(* CoDeSys 2.3.9.35 project: Q4_SISTEMA_DE_ESTEIRA_(COM MODELO).pro *)
(* Author: Altus *)
(* Libraries: DU35x.lib 7.7.11 15:59:13, Navigation.lib 15.7.11 10:06:00, SysLibTargetVisu.lib 26.11.08 09:53:28, Standard.lib 26.11.08 09:46:20, Iecsfc.lib 26.11.08 09:46:14, SYSLIBCALLBACK.LIB 26.11.08 09:53:30 *)

(* PLC configuration (modules and I/O channels)
Configuração do CP [Root] node -1, in %IB0 out %QB0
  Comunicação [Comunica] node 0, in %IB0 out %QB0
    COM1 [COM1] node 0, in %IB0 out %QB0 {BaudRate = 115200; Paridade = Sem Paridade; StopBits = 1 Stop Bit; Modem = Sem RTS/CTS; Delay = 5}
      MToolIEC [Codesys] node 0, in %IB0 out %QB0
    COM2 [COM2] node 1, in %IB0 out %QB0 {BaudRate = 115200; Paridade = Sem Paridade; StopBits = 1 Stop Bit; Modem = Sem RTS/CTS; Delay = 5}
      Desabilitada [Desabilitado485] node 0, in %IB0 out %QB0
  Barramento [Barramento] node 1, in %IB0 out %QB0
    Entradas [Entradas] node 0, in %IB0 out %QB0
      Entradas Digitais 0 [Entradas0] node 0, in %IW0 out %QB0
        I00 AT %IX0.0 [BitInput] I0.0
        I01 AT %IX0.1 [BitInput] I0.1
        I02 AT %IX0.2 [BitInput] I0.2
        I03 AT %IX0.3 [BitInput] I0.3
        I04 AT %IX0.4 [BitInput] I0.4
        I05 AT %IX0.5 [BitInput] I0.5
        I06 AT %IX0.6 [BitInput] I0.6
        I07 AT %IX0.7 [BitInput] I0.7
        I08 AT %IX0.8 [BitInput] I0.8
      Entradas Digitais 1 [Entradas1] node 0, in %IW1 out %QB0
        I10 AT %IX1.0 [BitInput] I1.0
        I11 AT %IX1.1 [BitInput] I1.1
        I12 AT %IX1.2 [BitInput] I1.2
        I13 AT %IX1.3 [BitInput] I1.3
        I14 AT %IX1.4 [BitInput] I1.4
        I15 AT %IX1.5 [BitInput] I1.5
        I16 AT %IX1.6 [BitInput] I1.6
        I17 AT %IX1.7 [BitInput] I1.7
        I18 AT %IX1.8 [BitInput] I1.8
      Entradas Digitais 2 [Entradas2] node 0, in %IW2 out %QB0
        I20 AT %IX2.0 [BitInput] I2.0
        I21 AT %IX2.1 [BitInput] I2.1
      Entradas Analógicas [EntradaAnalogica] node 0, in %IW4 out %QB0
        AI0 AT %IW4 [WordInput] AI0 {TipoAnalogica = Channel Disable; FiltroAnalogica = Filter 0 - AI=2ms  / AV=90ms; FundoEscala = 0}
        AI1 AT %IW5 [WordInput] AI1 {TipoAnalogica = Channel Disable; FiltroAnalogica = Filter 0 - AI=2ms  / AV=90ms; FundoEscala = 0}
        AI2 AT %IW6 [WordInput] AI2 {TipoAnalogica = Channel Disable; FiltroAnalogica = Filter 0 - AI=2ms  / AV=90ms; FundoEscala = 0}
        AI3 AT %IW7 [WordInput] AI3 {TipoAnalogica = Channel Disable; FiltroAnalogica = Filter 0 - AI=2ms  / AV=90ms; FundoEscala = 0}
      Entradas Rápidas [EntradasRapidas] node 1, in %IB16 out %QB0
        Bloco 0 [Bloco0] node 0, in %IB16 out %QB0
          Desabilitado [DesabilitadoBloco0] node 0, in %IB16 out %QB0
        Bloco 1 [Bloco1] node 1, in %IB16 out %QB0
          Desabilitado [DesabilitadoBloco1] node 0, in %IB16 out %QB0
        Entrada Configuravél Bloco 0 [EntradaConfiBloco0] node 2, in %IB16 out %QB0
          Contador 0 [EntradaConfContador0] node 0, in %IB16 out %QB0 {EntradaConfiguravelContador = Disable}
        Entrada Configuravél Bloco 1 [EntradaConfiBloco1] node 3, in %IB16 out %QB0
          Contador 2 [EntradaConfContador2] node 0, in %IB16 out %QB0 {EntradaConfiguravelContador = Disable}
    Saídas [Saidas] node 1, in %IB13 out %QB0
      Saídas Digitais 0 [Saidas0] node 0, in %IW0 out %QW0
        Q00 AT %QX0.0 [BitOutput] Q0.0
        Q01 AT %QX0.1 [BitOutput] Q0.1
        Q02 AT %QX0.2 [BitOutput] Q0.2
        Q03 AT %QX0.3 [BitOutput] Q0.3
        Q04 AT %QX0.4 [BitOutput] Q0.4
        Q05 AT %QX0.5 [BitOutput] Q0.5
        Q06 AT %QX0.6 [BitOutput] Q0.6
        Q07 AT %QX0.7 [BitOutput] Q0.7
      Saídas Digitais 1 [Saidas1] node 0, in %IW0 out %QW1
        Q10 AT %QX1.0 [BitOutput] Q1.0
        Q11 AT %QX1.1 [BitOutput] Q1.1
        Q12 AT %QX1.2 [BitOutput] Q1.2
        Q13 AT %QX1.3 [BitOutput] Q1.3
        Q14 AT %QX1.4 [BitOutput] Q1.4
        Q15 AT %QX1.5 [BitOutput] Q1.5
        Q16 AT %QX1.6 [BitOutput] Q1.6
        Q17 AT %QX1.7 [BitOutput] Q1.7
      Saídas Analógicas [SaidaAnalogica] node 0, in %IW0 out %QW3
        AO0 AT %QW3 [WordOutput] AO0 {TipoAnalogica = Channel Disable; FundoEscala = 0}
        AO1 AT %QW4 [WordOutput] AO1 {TipoAnalogica = Channel Disable; FundoEscala = 0}
      Saídas Rápidas [SaidasRapidas] node 1, in %IB0 out %QB10
        Saída Rápida 0 Desabilitada [DesabilitadoF0] node 0, in %IB0 out %QB10
        Saída Rápida 1 Desabilitada [DesabilitadoF1] node 1, in %IB0 out %QB10
      Saídas Comum de Contador [SaidasContador] node 2, in %IB0 out %QB10
        Saída do Bloco 0 Desabilitada [DesabilitadoSaidaBloco0] node 0, in %IB0 out %QB10
        Saída do Bloco 1 Desabilitada [DesabilitadoSaidaBloco1] node 1, in %IB0 out %QB10
  Eventos Externos [Eventos] node 2, in %IB13 out %QB6
    Evento Temporizado [TimerEvent] node 0, in %IB13 out %QB6 {Intervalo = 10}
*)

(* Task configuration *)
TASK PRINCIPAL (PRIORITY := 1, INTERVAL := T#1ms);
	PLC_PRG();
END_TASK
TASK NAVIGATION (PRIORITY := 1, INTERVAL := T#20ms);
	NAVEGA();
END_TASK
TASK VISUALIZATION (PRIORITY := 1, INTERVAL := T#500ms);
	MAINTARGETVISU_PAINT_CODE
END_TASK
TASK KEYBOARD_USAGE (PRIORITY := 1, INTERVAL := T#20ms);
	MAINTARGETVISU_INPUT_CODE
END_TASK

(* POU PLC_PRG, LD *)
PROGRAM PLC_PRG
VAR
    (* ========================================================= *)
    (* ENTRADAS FISICAS (Chaves e Sensores - %IX)             *)
    (* ========================================================= *)
    a0 AT %IX0.0: BOOL; (* Sensor de Fim de Curso: Cilindro A Recuado *)
    a1 AT %IX0.1: BOOL; (* Sensor de Fim de Curso: Cilindro A Avancado *)
    b0 AT %IX0.2: BOOL; (* Sensor de Fim de Curso: Cilindro B Recuado *)
    b1 AT %IX0.3: BOOL; (* Sensor de Fim de Curso: Cilindro B Avancado *)
    c0 AT %IX0.4: BOOL; (* Sensor de Fim de Curso: Cilindro C Recuado *)
    c1 AT %IX0.5: BOOL; (* Sensor de Fim de Curso: Cilindro C Avancado *)
    CH AT %IX0.6: BOOL; (* Chave de Controle de Ciclo S *)
    SP AT %IX0.7: BOOL; (* Sensor de Presenca de Embalagem Sp - NF *)

    (* ========================================================= *)
    (* SAIDAS FISICAS (Atuadores - %QX)                       *)
    (* ========================================================= *)
    CA AT %QX1.0: BOOL; (* Comando: Valvula do Cilindro A *)
    CB AT %QX1.1: BOOL; (* Comando: Valvula do Cilindro B *)
    CC AT %QX1.2: BOOL; (* Comando: Valvula do Cilindro C *)
    M  AT %QX1.3: BOOL; (* Comando: Motor de acionamento da esteira *)

    (* ========================================================= *)
    (* ESTADOS DO AFD (Memorias de Etapa - %MX1.x)            *)
    (* ========================================================= *)
    S0 AT %MX1.0: BOOL; (* Estado 0: Repouso / Espera de embalagem *)
    S1 AT %MX1.1: BOOL; (* Estado 1: Avancar Cilindro A *)
    S2 AT %MX1.2: BOOL; (* Estado 2: Avancar Cilindro B *)
    S3 AT %MX1.3: BOOL; (* Estado 3: Recuar Cilindro C e Dosagem *)
    S4 AT %MX1.4: BOOL; (* Estado 4: Avancar Cilindro C *)
    S5 AT %MX1.5: BOOL; (* Estado 5: Recuar A e B simultaneamente *)
    S6 AT %MX1.6: BOOL; (* Estado 6: Esperar saida da embalagem cheia *)
    S_erro AT %MX1.7: BOOL; (* Estado Erro: Seguranca e Intertravamento *)

    (* ========================================================= *)
    (* TRANSICOES DO AFD (Condicoes de Disparo - %MX2.x e %MX3.x)*)
    (* ========================================================= *)
    T0 AT %MX2.0: BOOL; (* Disparo da transicao de S0 para S1 *)
    T1 AT %MX2.1: BOOL; (* Disparo da transicao de S1 para S2 *)
    T2 AT %MX2.2: BOOL; (* Disparo da transicao de S2 para S3 *)
    T3 AT %MX2.3: BOOL; (* Disparo da transicao de S3 para S4 *)
    T4 AT %MX2.4: BOOL; (* Disparo da transicao de S4 para S5 *)
    T5 AT %MX2.5: BOOL; (* Disparo da transicao de S5 para S6 *)
    T6 AT %MX2.6: BOOL; (* Disparo da transicao de S6 para S0 *)
    TE AT %MX3.2: BOOL; (* Disparo da transicao Global de Falha para S_erro *)
    TR AT %MX3.1: BOOL; (* Disparo da transicao de Retorno para S0 *)

    (* ========================================================= *)
    (* VARIAVEIS INTERNAS DE CONTROLO E SINALIZACAO           *)
    (* ========================================================= *)
    F      AT %MX0.6: BOOL; (* Flag: Condicao Global de Falha Ativa *)
    RESET  AT %MX3.0: BOOL; (* Comando/Flag de Reset de Erro *)
    ALARME AT %MX3.4: BOOL; (* Sinalizacao de Alarme / Intertravamento *)

    (* ========================================================= *)
    (* BLOCO FUNCIONAL: TEMPORIZADOR (Dosagem)                *)
    (* ========================================================= *)
    TEMPORIZADOR1: TON;     (* Instancia do Bloco Timer On-Delay *)
    T1_EN AT %MX0.2: BOOL;  (* Sinal para habilitar/iniciar a contagem do tempo *)
    QT1   AT %MX0.3: BOOL;  (* Saida de tempo esgotado 5 segundos *)

    (* ========================================================= *)
    (* BLOCO FUNCIONAL: CONTADOR (Lote de 10 Ciclos)          *)
    (* ========================================================= *)
    CTU: CTU;         (* CORRIGIDO: Nao usar CTU: CTU para evitar erro *)
    CU    AT %MX0.0: BOOL;  (* Pulso de entrada para incremento do contador *)
    QCU   AT %MX0.1: BOOL;  (* Saida indicando que o limite do lote foi atingido *)
    COUNT AT %MW10: INT;    (* Registo de memoria Word com o valor atual *)
    P: R_TRIG;              (* Bloco detetor de borda de subida Trigger *)
END_VAR
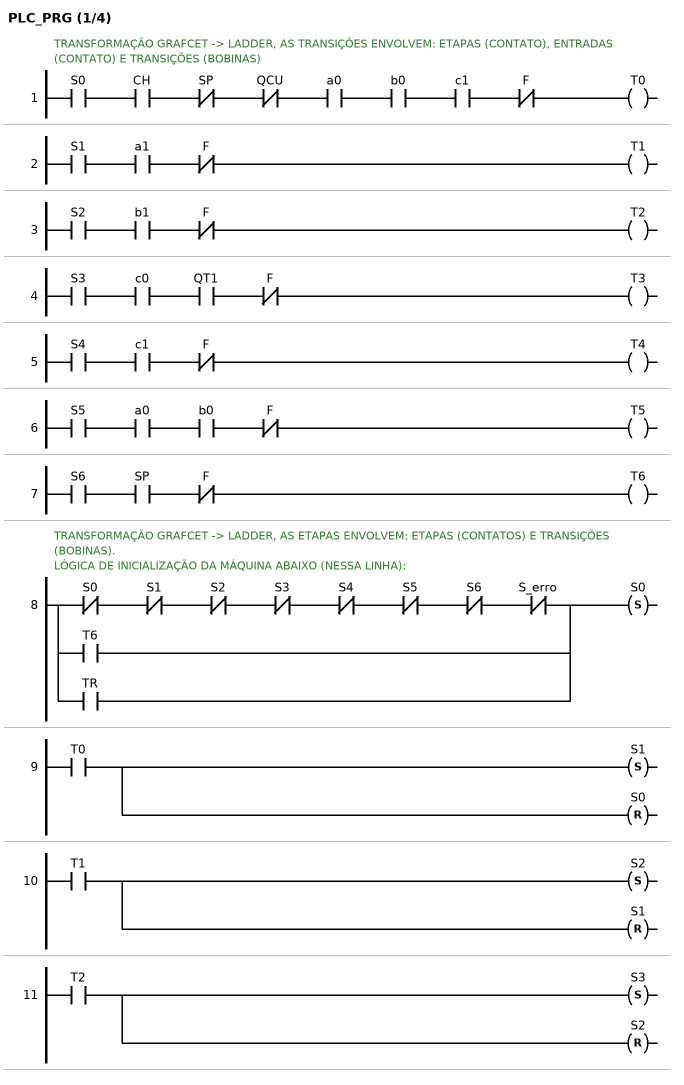
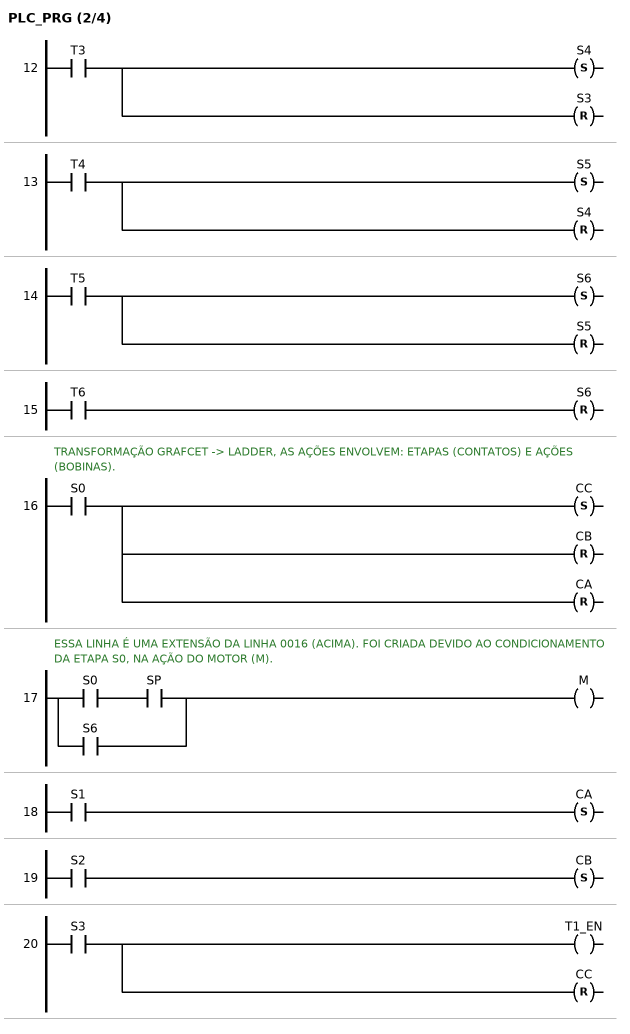
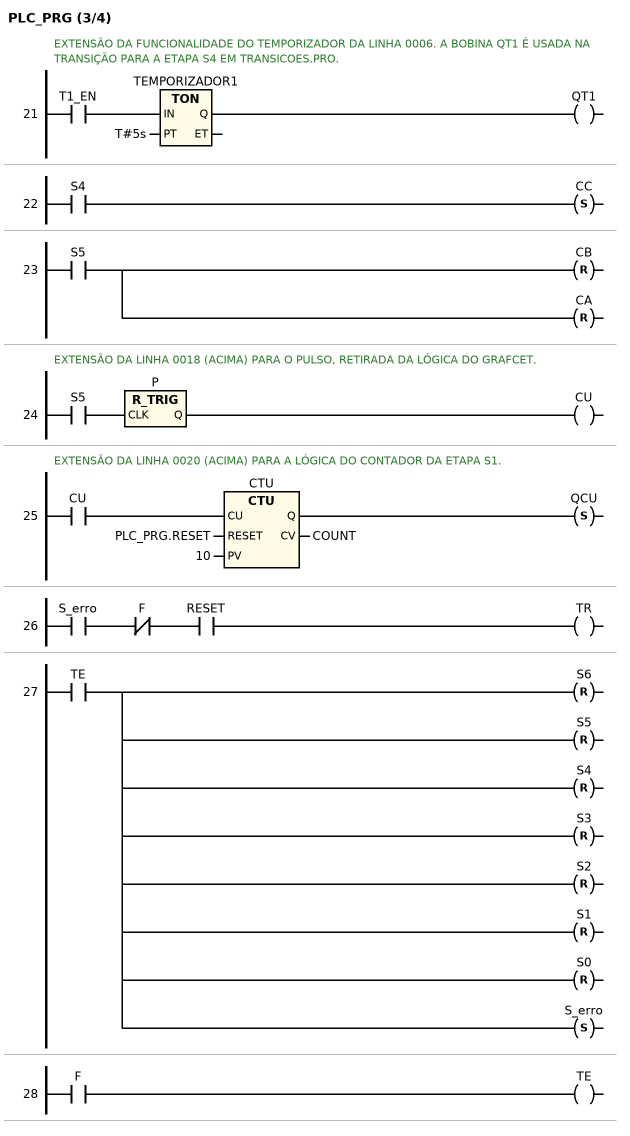
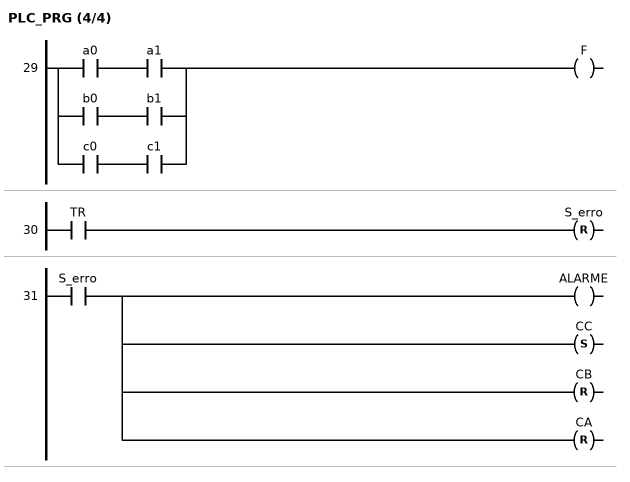
_LD_ (* Ladder Diagram *)
NETWORK 1 (* TRANSFORMAÇÃO GRAFCET -> LADDER, AS TRANSIÇÕES ENVOLVEM: ETAPAS (CONTATO), ENTRADAS (CONTATO) E TRANSIÇÕES (BOBINAS) *)
	[S0] - [CH] - [/SP] - [/QCU] - [a0] - [b0] - [c1] - [/F] --- (T0)
NETWORK 2
	[S1] - [a1] - [/F] --- (T1)
NETWORK 3
	[S2] - [b1] - [/F] --- (T2)
NETWORK 4
	[S3] - [c0] - [QT1] - [/F] --- (T3)
NETWORK 5
	[S4] - [c1] - [/F] --- (T4)
NETWORK 6
	[S5] - [a0] - [b0] - [/F] --- (T5)
NETWORK 7
	[S6] - [SP] - [/F] --- (T6)
NETWORK 8 (* TRANSFORMAÇÃO GRAFCET -> LADDER, AS ETAPAS ENVOLVEM: ETAPAS (CONTATOS) E TRANSIÇÕES (BOBINAS). / LÓGICA DE INICIALIZAÇÃO DA MÁQUINA ABAIXO (NESSA LINHA): *)
	{ [/S0] - [/S1] - [/S2] - [/S3] - [/S4] - [/S5] - [/S6] - [/S_erro] | [T6] | [TR] } --- (S S0)
NETWORK 9
	[T0] --- (S S1) (R S0)
NETWORK 10
	[T1] --- (S S2) (R S1)
NETWORK 11
	[T2] --- (S S3) (R S2)
NETWORK 12
	[T3] --- (S S4) (R S3)
NETWORK 13
	[T4] --- (S S5) (R S4)
NETWORK 14
	[T5] --- (S S6) (R S5)
NETWORK 15
	[T6] --- (R S6)
NETWORK 16 (* TRANSFORMAÇÃO GRAFCET -> LADDER, AS AÇÕES ENVOLVEM: ETAPAS (CONTATOS) E AÇÕES (BOBINAS). *)
	[S0] --- (S CC) (R CB) (R CA)
NETWORK 17 (* ESSA LINHA É UMA EXTENSÃO DA LINHA 0016 (ACIMA). FOI CRIADA DEVIDO AO CONDICIONAMENTO DA ETAPA S0, NA AÇÃO DO MOTOR (M). *)
	{ [S0] - [SP] | [S6] } --- (M)
NETWORK 18
	[S1] --- (S CA)
NETWORK 19
	[S2] --- (S CB)
NETWORK 20
	[S3] --- (T1_EN) (R CC)
NETWORK 21 (* EXTENSÃO DA FUNCIONALIDADE DO TEMPORIZADOR DA LINHA 0006. A BOBINA QT1 É USADA NA TRANSIÇÃO PARA A ETAPA S4 EM TRANSICOES.PRO. *)
	[T1_EN] - TEMPORIZADOR1:TON(IN: *, PT: T#5s) --- (QT1)
NETWORK 22
	[S4] --- (S CC)
NETWORK 23
	[S5] --- (R CB) (R CA)
NETWORK 24 (* EXTENSÃO DA LINHA 0018 (ACIMA) PARA O PULSO, RETIRADA DA LÓGICA DO GRAFCET. *)
	[S5] - P:R_TRIG(CLK: *) --- (CU)
NETWORK 25 (* EXTENSÃO DA LINHA 0020 (ACIMA) PARA A LÓGICA DO CONTADOR DA ETAPA S1. *)
	[CU] - CTU:CTU(CU: *, RESET: PLC_PRG.RESET, PV: 10, CV => COUNT) --- (S QCU)
NETWORK 26
	[S_erro] - [/F] - [RESET] --- (TR)
NETWORK 27
	[TE] --- (R S6) (R S5) (R S4) (R S3) (R S2) (R S1) (R S0) (S S_erro)
NETWORK 28
	[F] --- (TE)
NETWORK 29
	{ [a0] - [a1] | [b0] - [b1] | [c0] - [c1] } --- (F)
NETWORK 30
	[TR] --- (R S_erro)
NETWORK 31
	[S_erro] --- (ALARME) (S CC) (R CB) (R CA)
_END_LD_
(* the same logic as Structured Text *)
(* Network 1: TRANSFORMAÇÃO GRAFCET -> LADDER, AS TRANSIÇÕES ENVOLVEM: ETAPAS (CONTATO), ENTRADAS (CONTATO) E TRANSIÇÕES (BOBINAS) *)
T0 := S0 AND CH AND NOT SP AND NOT QCU AND a0 AND b0 AND c1 AND NOT F;
(* Network 2 *)
T1 := S1 AND a1 AND NOT F;
(* Network 3 *)
T2 := S2 AND b1 AND NOT F;
(* Network 4 *)
T3 := S3 AND c0 AND QT1 AND NOT F;
(* Network 5 *)
T4 := S4 AND c1 AND NOT F;
(* Network 6 *)
T5 := S5 AND a0 AND b0 AND NOT F;
(* Network 7 *)
T6 := S6 AND SP AND NOT F;
(* Network 8: TRANSFORMAÇÃO GRAFCET -> LADDER, AS ETAPAS ENVOLVEM: ETAPAS (CONTATOS) E TRANSIÇÕES (BOBINAS). / LÓGICA DE INICIALIZAÇÃO DA MÁQUINA ABAIXO (NESSA LINHA): *)
IF NOT S0 AND NOT S1 AND NOT S2 AND NOT S3 AND NOT S4 AND NOT S5 AND NOT S6 AND NOT S_erro OR T6 OR TR THEN S0 := TRUE; END_IF;
(* Network 9 *)
IF T0 THEN S1 := TRUE; S0 := FALSE; END_IF;
(* Network 10 *)
IF T1 THEN S2 := TRUE; S1 := FALSE; END_IF;
(* Network 11 *)
IF T2 THEN S3 := TRUE; S2 := FALSE; END_IF;
(* Network 12 *)
IF T3 THEN S4 := TRUE; S3 := FALSE; END_IF;
(* Network 13 *)
IF T4 THEN S5 := TRUE; S4 := FALSE; END_IF;
(* Network 14 *)
IF T5 THEN S6 := TRUE; S5 := FALSE; END_IF;
(* Network 15 *)
IF T6 THEN S6 := FALSE; END_IF;
(* Network 16: TRANSFORMAÇÃO GRAFCET -> LADDER, AS AÇÕES ENVOLVEM: ETAPAS (CONTATOS) E AÇÕES (BOBINAS). *)
IF S0 THEN CC := TRUE; CB := FALSE; CA := FALSE; END_IF;
(* Network 17: ESSA LINHA É UMA EXTENSÃO DA LINHA 0016 (ACIMA). FOI CRIADA DEVIDO AO CONDICIONAMENTO DA ETAPA S0, NA AÇÃO DO MOTOR (M). *)
M := S0 AND SP OR S6;
(* Network 18 *)
IF S1 THEN CA := TRUE; END_IF;
(* Network 19 *)
IF S2 THEN CB := TRUE; END_IF;
(* Network 20 *)
T1_EN := S3;
IF S3 THEN CC := FALSE; END_IF;
(* Network 21: EXTENSÃO DA FUNCIONALIDADE DO TEMPORIZADOR DA LINHA 0006. A BOBINA QT1 É USADA NA TRANSIÇÃO PARA A ETAPA S4 EM TRANSICOES.PRO. *)
TEMPORIZADOR1(IN := T1_EN, PT := T#5s);
QT1 := TEMPORIZADOR1.Q;
(* Network 22 *)
IF S4 THEN CC := TRUE; END_IF;
(* Network 23 *)
IF S5 THEN CB := FALSE; CA := FALSE; END_IF;
(* Network 24: EXTENSÃO DA LINHA 0018 (ACIMA) PARA O PULSO, RETIRADA DA LÓGICA DO GRAFCET. *)
P(CLK := S5);
CU := P.Q;
(* Network 25: EXTENSÃO DA LINHA 0020 (ACIMA) PARA A LÓGICA DO CONTADOR DA ETAPA S1. *)
CTU(CU := CU, RESET := PLC_PRG.RESET, PV := 10);
COUNT := CTU.CV;
IF CTU.Q THEN QCU := TRUE; END_IF;
(* Network 26 *)
TR := S_erro AND NOT F AND RESET;
(* Network 27 *)
IF TE THEN S6 := FALSE; S5 := FALSE; S4 := FALSE; S3 := FALSE; S2 := FALSE; S1 := FALSE; S0 := FALSE; S_erro := TRUE; END_IF;
(* Network 28 *)
TE := F;
(* Network 29 *)
F := a0 AND a1 OR b0 AND b1 OR c0 AND c1;
(* Network 30 *)
IF TR THEN S_erro := FALSE; END_IF;
(* Network 31 *)
ALARME := S_erro;
IF S_erro THEN CC := TRUE; END_IF;
IF S_erro THEN CB := FALSE; END_IF;
IF S_erro THEN CA := FALSE; END_IF;
END_PROGRAM
ACTION ACOES:
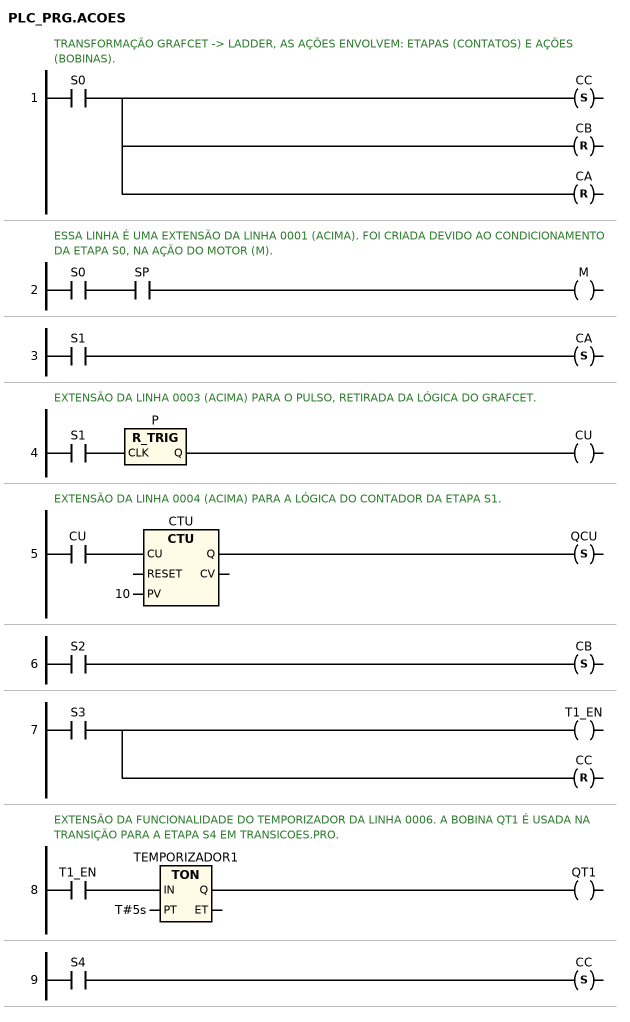
_LD_ (* Ladder Diagram *)
NETWORK 1 (* TRANSFORMAÇÃO GRAFCET -> LADDER, AS AÇÕES ENVOLVEM: ETAPAS (CONTATOS) E AÇÕES (BOBINAS). *)
	[S0] --- (S CC) (R CB) (R CA)
NETWORK 2 (* ESSA LINHA É UMA EXTENSÃO DA LINHA 0001 (ACIMA). FOI CRIADA DEVIDO AO CONDICIONAMENTO DA ETAPA S0, NA AÇÃO DO MOTOR (M). *)
	[S0] - [SP] --- (M)
NETWORK 3
	[S1] --- (S CA)
NETWORK 4 (* EXTENSÃO DA LINHA 0003 (ACIMA) PARA O PULSO, RETIRADA DA LÓGICA DO GRAFCET. *)
	[S1] - P:R_TRIG(CLK: *) --- (CU)
NETWORK 5 (* EXTENSÃO DA LINHA 0004 (ACIMA) PARA A LÓGICA DO CONTADOR DA ETAPA S1. *)
	[CU] - CTU:CTU(CU: *, RESET: , PV: 10) --- (S QCU)
NETWORK 6
	[S2] --- (S CB)
NETWORK 7
	[S3] --- (T1_EN) (R CC)
NETWORK 8 (* EXTENSÃO DA FUNCIONALIDADE DO TEMPORIZADOR DA LINHA 0006. A BOBINA QT1 É USADA NA TRANSIÇÃO PARA A ETAPA S4 EM TRANSICOES.PRO. *)
	[T1_EN] - TEMPORIZADOR1:TON(IN: *, PT: T#5s) --- (QT1)
NETWORK 9
	[S4] --- (S CC)
_END_LD_
(* the same logic as Structured Text *)
(* Network 1 *)
IF S0 THEN CC := TRUE; CB := FALSE; CA := FALSE; END_IF;
(* Network 2 *)
M := S0 AND SP;
(* Network 3 *)
IF S1 THEN CA := TRUE; END_IF;
(* Network 4 *)
P(CLK := S1);
CU := P.Q;
(* Network 5: see the listing above *)
(* Network 6 *)
IF S2 THEN CB := TRUE; END_IF;
(* Network 7 *)
T1_EN := S3;
IF S3 THEN CC := FALSE; END_IF;
(* Network 8 *)
TEMPORIZADOR1(IN := T1_EN, PT := T#5s);
QT1 := TEMPORIZADOR1.Q;
(* Network 9 *)
IF S4 THEN CC := TRUE; END_IF;
END_ACTION
ACTION ETAPAS:
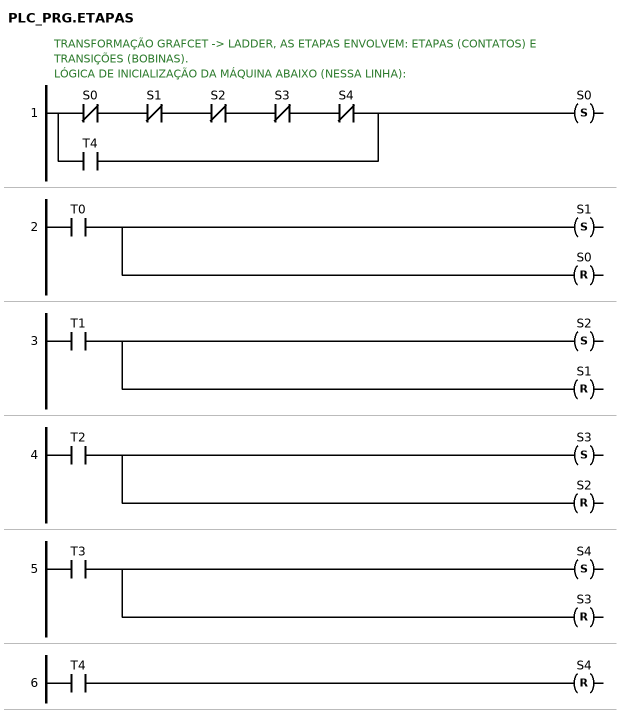
_LD_ (* Ladder Diagram *)
NETWORK 1 (* TRANSFORMAÇÃO GRAFCET -> LADDER, AS ETAPAS ENVOLVEM: ETAPAS (CONTATOS) E TRANSIÇÕES (BOBINAS). / LÓGICA DE INICIALIZAÇÃO DA MÁQUINA ABAIXO (NESSA LINHA): *)
	{ [/S0] - [/S1] - [/S2] - [/S3] - [/S4] | [T4] } --- (S S0)
NETWORK 2
	[T0] --- (S S1) (R S0)
NETWORK 3
	[T1] --- (S S2) (R S1)
NETWORK 4
	[T2] --- (S S3) (R S2)
NETWORK 5
	[T3] --- (S S4) (R S3)
NETWORK 6
	[T4] --- (R S4)
_END_LD_
(* the same logic as Structured Text *)
(* Network 1: TRANSFORMAÇÃO GRAFCET -> LADDER, AS ETAPAS ENVOLVEM: ETAPAS (CONTATOS) E TRANSIÇÕES (BOBINAS). / LÓGICA DE INICIALIZAÇÃO DA MÁQUINA ABAIXO (NESSA LINHA): *)
IF NOT S0 AND NOT S1 AND NOT S2 AND NOT S3 AND NOT S4 OR T4 THEN S0 := TRUE; END_IF;
(* Network 2 *)
IF T0 THEN S1 := TRUE; S0 := FALSE; END_IF;
(* Network 3 *)
IF T1 THEN S2 := TRUE; S1 := FALSE; END_IF;
(* Network 4 *)
IF T2 THEN S3 := TRUE; S2 := FALSE; END_IF;
(* Network 5 *)
IF T3 THEN S4 := TRUE; S3 := FALSE; END_IF;
(* Network 6 *)
IF T4 THEN S4 := FALSE; END_IF;
END_ACTION
ACTION TRANSICOES:
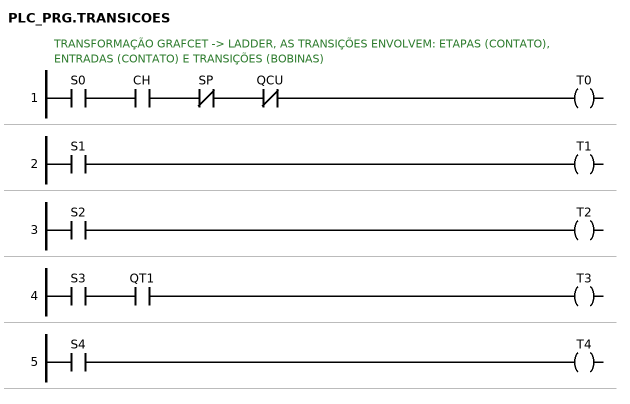
_LD_ (* Ladder Diagram *)
NETWORK 1 (* TRANSFORMAÇÃO GRAFCET -> LADDER, AS TRANSIÇÕES ENVOLVEM: ETAPAS (CONTATO), ENTRADAS (CONTATO) E TRANSIÇÕES (BOBINAS) *)
	[S0] - [CH] - [/SP] - [/QCU] --- (T0)
NETWORK 2
	[S1] --- (T1)
NETWORK 3
	[S2] --- (T2)
NETWORK 4
	[S3] - [QT1] --- (T3)
NETWORK 5
	[S4] --- (T4)
_END_LD_
(* the same logic as Structured Text *)
(* Network 1: TRANSFORMAÇÃO GRAFCET -> LADDER, AS TRANSIÇÕES ENVOLVEM: ETAPAS (CONTATO), ENTRADAS (CONTATO) E TRANSIÇÕES (BOBINAS) *)
T0 := S0 AND CH AND NOT SP AND NOT QCU;
(* Network 2 *)
T1 := S1;
(* Network 3 *)
T2 := S2;
(* Network 4 *)
T3 := S3 AND QT1;
(* Network 5 *)
T4 := S4;
END_ACTION

(* POU NAVEGA, ST *)
PROGRAM NAVEGA
VAR
	ControleTelas : NAVIGATION;
	ListaTelas 	: ARRAY [0..30] OF STRING(10);
END_VAR
(* Adiciona a tela MAIN como tela principal *)
ListaTelas[0] := 'MAIN';

(* Ativa o controle automático de navegação somente pelo teclado *)
ControleTelas(ENABLE_UPDW := FALSE, VISU_LIST := ListaTelas, UP := FALSE , DOWN := FALSE);
END_PROGRAM

(* Visualisation V1
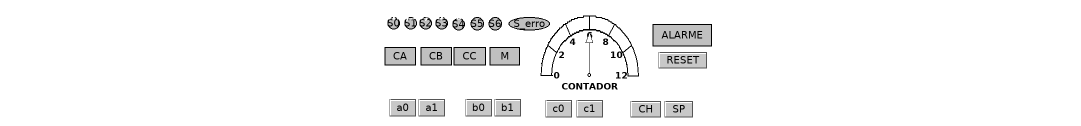
button at (250,88)-(280,104): text "CH"; toggles PLC_PRG.CH
button at (284,88)-(312,104): text "SP"; toggles PLC_PRG.SP
ellipse at (7,4)-(19,16): text "S0"; alarm colour if PLC_PRG.S0
ellipse at (24,4)-(36,16): text "S1"; alarm colour if PLC_PRG.S1
ellipse at (39,4)-(51,16): text "S2"; alarm colour if PLC_PRG.S2
ellipse at (55,4)-(67,16): text "S3"; alarm colour if PLC_PRG.S3
ellipse at (72,5)-(84,17): text "S4"; alarm colour if PLC_PRG.S4
group at (159,2)-(258,82)
  rectangle at (0,0)-(1,1): text "{ExtendedElement},Visu\ElementDLL.ete,0,@Zeigerinstrument,99,180,0,0,255,255,255,0,PLC_PRG.COUNT,CONTADOR,%.0f,1,1,1,2,2,0,12,0,0,0,0,0,0,0,-11,80,700,Arial,1,0,"
  rectangle at (14,43)-(20,57): text "0"
  rectangle at (19,26)-(25,40): text "2"
  rectangle at (30,15)-(36,29): text "4"
  rectangle at (47,10)-(53,24): text "6"
  rectangle at (63,15)-(69,29): text "8"
  rectangle at (71,26)-(83,40): text "10"
  rectangle at (76,43)-(88,57): text "12"
  rectangle at (20,52)-(80,66): text "CONTADOR"
  polygon at (46,14)-(53,50): angle ((PLC_PRG.COUNT * 1.0)-6) * 15
ellipse at (90,4)-(103,17): text "S5"; alarm colour if PLC_PRG.S5
button at (9,86)-(35,103): text "a0"; toggles PLC_PRG.a0
button at (38,86)-(64,103): text "a1"; toggles PLC_PRG.a1
button at (85,86)-(111,103): text "b0"; toggles PLC_PRG.b0
button at (114,86)-(140,103): text "b1"; toggles PLC_PRG.b1
button at (165,87)-(191,104): text "c0"; toggles PLC_PRG.c0
button at (196,87)-(222,104): text "c1"; toggles PLC_PRG.c1
rectangle at (272,11)-(331,33): text "ALARME"; alarm colour if PLC_PRG.ALARME
ellipse at (108,4)-(121,17): text "S6"; alarm colour if PLC_PRG.S6
rectangle at (4,34)-(35,52): text "CA"; alarm colour if PLC_PRG.CA
rectangle at (40,34)-(71,52): text "CB"; alarm colour if PLC_PRG.CB
rectangle at (73,34)-(105,52): text "CC"; alarm colour if PLC_PRG.CC
rectangle at (109,34)-(139,52): text "M"; alarm colour if PLC_PRG.M
ellipse at (128,4)-(169,17): text "S_erro"; alarm colour if PLC_PRG.S_erro
button at (278,39)-(326,55): text "RESET"; toggles PLC_PRG.RESET
10 more shapes without text or variables
*)
